SUBAPPLICATION E_PERMIT_INVERT (* Invertiertes Event-Freigabe-Gate (F_NOT_BOOL_INIT + E_PERMIT) *)
  (* Standard: 61499-2; Description: Copyright (c) 2026 Meisterschulen am Ostbahnhof This program and the accompanying materials are made available under the terms of the Eclipse Public License 2.0 which is available at https://www.eclipse.org/legal/epl-2.0/ SPDX-License-Identifier: EPL-2.0 *)
  (* Version 1.0, 2026-09-10, Franz Höpfinger, Meisterschulen am Ostbahnhof, initial implementation *)
  PACKAGE MyLib::sys;
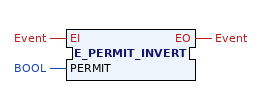
  EVENT_INPUT
    EI; (* Event input (wird durchgelassen wenn PERMIT FALSE ist) *)
  END_EVENT
  EVENT_OUTPUT
    EO; (* Event output (feuert wenn EI eintrifft und PERMIT FALSE ist) *)
  END_EVENT
  VAR_INPUT
    PERMIT : BOOL; (* Invertierte Freigabebedingung *)
  END_VAR
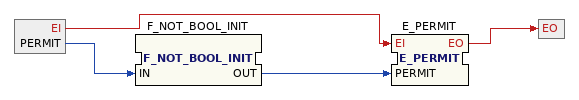
  FBS
    F_NOT_BOOL_INIT : iec61131::booleanOperators::F_NOT_BOOL_INIT;
    E_PERMIT : iec61499::events::E_PERMIT;
  END_FBS
  EVENT_CONNECTIONS
    EI TO E_PERMIT.EI;
    E_PERMIT.EO TO EO;
  END_CONNECTIONS
  DATA_CONNECTIONS
    PERMIT TO F_NOT_BOOL_INIT.IN;
    F_NOT_BOOL_INIT.OUT TO E_PERMIT.PERMIT;
  END_CONNECTIONS
END_SUBAPPLICATION
